FUNCTION_BLOCK FB_GC EXTENDS FB_PackMLModeSet
VAR_INPUT
	ServiceCtrl : REFERENCE TO ST_GC_ServiceCtrl;
	ServiceStatus : REFERENCE TO ST_GC_ServiceStatus;
	Admin : REFERENCE TO ST_GC_Admin;
	
	// Base unit used in GC chamber
	SpinAxis_BaseUnit : REFERENCE TO FB_AxisControl;
END_VAR

VAR_OUTPUT
	
END_VAR

VAR
	// 有需要特殊操作的需求，所以建立一個 ST_GC_ServiceCtrl 變數，讓程式內部可以過一手處理
	_ServiceCtrl : ST_GC_ServiceCtrl;
	_SpinAxisJogService : FB_GCSpinAxisJogServices;
	_SpinAxisMoveAbsService : FB_GCSpinAxisMoveAbsServices;
	_SpinAxisMoveVelService : FB_GCSpinAxisMoveVelServices;
END_VAR

A00_Service();
SUPER^();

ACTION A00_Service:
_SpinAxisJogService(
	Ctrl:= _ServiceCtrl.SpinAxisJog,
	Status:= ServiceStatus.SpinAxisJog,
	Axis_BaseUnit:= SpinAxis_BaseUnit,
	// Owner IDs are assigned by the Module so each Service instance is unique.
	ResourceOwnerId:= E_GCResourceOwnerId.SpinAxisJog);

_SpinAxisMoveAbsService(
	Ctrl:= _ServiceCtrl.SpinAxisMoveAbs,
	Status:= ServiceStatus.SpinAxisMoveAbs,
	Axis_BaseUnit:= SpinAxis_BaseUnit,
	ResourceOwnerId:= E_GCResourceOwnerId.SpinAxisMoveAbs);

_SpinAxisMoveVelService(
	Ctrl:= _ServiceCtrl.SpinAxisMoveVel,
	Status:= ServiceStatus.SpinAxisMoveVel,
	Axis_BaseUnit:= SpinAxis_BaseUnit,
	ResourceOwnerId:= E_GCResourceOwnerId.SpinAxisMoveVel);
END_ACTION

METHOD PROTECTED H_OnAborted
VAR_INPUT
	bFirstScan	: BOOL;
END_VAR
// Default action hook intentionally empty. Override in derived FBs when needed.
END_METHOD

METHOD PROTECTED H_OnAborting : E_PackMLHookResult
VAR_INPUT
	bFirstScan	: BOOL;
END_VAR
// Default transient hooks complete immediately; override when work is required.
H_OnAborting := E_PackMLHookResult.Done;
END_METHOD

METHOD PROTECTED H_OnClearing : E_PackMLHookResult
VAR_INPUT
	bFirstScan	: BOOL;
END_VAR
H_OnClearing := E_PackMLHookResult.Done;
END_METHOD

METHOD PROTECTED H_OnComplete
VAR_INPUT
	bFirstScan	: BOOL;
END_VAR
// Default action hook intentionally empty. Override in derived FBs when needed.
END_METHOD

METHOD PROTECTED H_OnCompleting : E_PackMLHookResult
VAR_INPUT
	bFirstScan	: BOOL;
END_VAR
// Default transient hooks complete immediately; override when work is required.
H_OnCompleting := E_PackMLHookResult.Done;
END_METHOD

METHOD PROTECTED H_OnExecute : E_PackMLHookResult
VAR_INPUT
	bFirstScan	: BOOL;
END_VAR
// Execute is stable by default; derived FBs decide when the process is done.
H_OnExecute := E_PackMLHookResult.Busy;

// Mapping control data
_ServiceCtrl := ServiceCtrl;
END_METHOD

METHOD PROTECTED H_OnHeld
VAR_INPUT
	bFirstScan	: BOOL;
END_VAR
// Default action hook intentionally empty. Override in derived FBs when needed.
END_METHOD

METHOD PROTECTED H_OnHolding : E_PackMLHookResult
VAR_INPUT
	bFirstScan	: BOOL;
END_VAR
// Default transient hooks complete immediately; override when work is required.
H_OnHolding := E_PackMLHookResult.Done;
END_METHOD

METHOD PROTECTED H_OnIdle
VAR_INPUT
	bFirstScan	: BOOL;
END_VAR
// Default action hook intentionally empty. Override in derived FBs when needed.
END_METHOD

METHOD PROTECTED H_OnModeChanged
VAR_INPUT
	ePreviousMode	: T_PackMLMode;
	eNewMode	: T_PackMLMode;
END_VAR
// Notice current mode to each service
_SpinAxisJogService.ModuleMode := eNewMode;
_SpinAxisMoveAbsService.ModuleMode := eNewMode;
_SpinAxisMoveVelService.ModuleMode := eNewMode;
END_METHOD

METHOD PROTECTED H_OnResetting : E_PackMLHookResult
VAR_INPUT
	bFirstScan	: BOOL;
END_VAR
H_OnResetting := E_PackMLHookResult.Busy;

// Request reset cmd to services
_ServiceCtrl.SpinAxisJog.Reset := TRUE;
_ServiceCtrl.SpinAxisMoveAbs.Reset := TRUE;
_ServiceCtrl.SpinAxisMoveVel.Reset := TRUE;

// Wait cmd finished
IF ServiceStatus.SpinAxisJog.State <> E_PackMLState.Idle
	OR ServiceStatus.SpinAxisMoveAbs.State <> E_PackMLState.Idle
	OR ServiceStatus.SpinAxisMoveVel.State <> E_PackMLState.Idle THEN
	RETURN;
END_IF

// Reset trigger
_ServiceCtrl.SpinAxisJog.Reset := FALSE;
_ServiceCtrl.SpinAxisMoveAbs.Reset := FALSE;
_ServiceCtrl.SpinAxisMoveVel.Reset := FALSE;

H_OnResetting := E_PackMLHookResult.Done;
END_METHOD

METHOD PROTECTED H_OnStarting : E_PackMLHookResult
VAR_INPUT
	bFirstScan	: BOOL;
END_VAR
// Default transient hooks complete immediately; override when work is required.
H_OnStarting := E_PackMLHookResult.Done;
END_METHOD

METHOD PROTECTED H_OnStopped
VAR_INPUT
	bFirstScan	: BOOL;
END_VAR
// Default action hook intentionally empty. Override in derived FBs when needed.
END_METHOD

METHOD PROTECTED H_OnStopping : E_PackMLHookResult
VAR_INPUT
	bFirstScan	: BOOL;
END_VAR
// Default transient hooks complete immediately; override when work is required.
H_OnStopping := E_PackMLHookResult.Done;
END_METHOD

METHOD PROTECTED H_OnSuspended
VAR_INPUT
	bFirstScan	: BOOL;
END_VAR
// Default action hook intentionally empty. Override in derived FBs when needed.
END_METHOD

METHOD PROTECTED H_OnSuspending : E_PackMLHookResult
VAR_INPUT
	bFirstScan	: BOOL;
END_VAR
// Default transient hooks complete immediately; override when work is required.
H_OnSuspending := E_PackMLHookResult.Done;
END_METHOD

METHOD PROTECTED H_OnUndefined : E_PackMLHookResult
VAR_INPUT
	bFirstScan	: BOOL;
END_VAR
// The base FB leaves Undefined immediately unless a derived FB delays startup.
H_OnUndefined := E_PackMLHookResult.Done;
END_METHOD

METHOD PROTECTED H_OnUnholding : E_PackMLHookResult
VAR_INPUT
	bFirstScan	: BOOL;
END_VAR
// Default transient hooks complete immediately; override when work is required.
H_OnUnholding := E_PackMLHookResult.Done;
END_METHOD

METHOD PROTECTED H_OnUnsuspending : E_PackMLHookResult
VAR_INPUT
	bFirstScan	: BOOL;
END_VAR
// Default transient hooks complete immediately; override when work is required.
H_OnUnsuspending := E_PackMLHookResult.Done;
END_METHOD

END_FUNCTION_BLOCK

(* stored: Version 1.1.0.1, ProductVersion 3.1.4026.18
   POU FB_GC: Id {d2b222b5-592d-46be-8a8e-fa50af509b93}, SpecialFunc None
   Folder StateAction: Id {92cfe23b-b998-4d76-8aa2-c8089e78aa61}
   Action A00_Service: Id {c62275db-aa76-4b4d-95ad-2ecb5851f919}
   Method H_OnAborted: Id {de8d6f56-427f-41df-b4d5-ddd289e1aed8}
   Method H_OnAborting: Id {29c05c7a-ae95-4991-b775-aae453451d8c}
   Method H_OnClearing: Id {b7069c3b-bd41-45c4-a177-00789e12f344}
   Method H_OnComplete: Id {9ab7169f-1450-41d3-b3d7-d608e72d68f0}
   Method H_OnCompleting: Id {6a295d34-cfdf-466f-b604-2e762f01df0b}
   Method H_OnExecute: Id {dc703a52-8c8a-4e2d-8deb-4adebb327ad6}
   Method H_OnHeld: Id {93f6b454-4398-4439-9237-4d01e13b7ccc}
   Method H_OnHolding: Id {d74d6d7d-e0fe-48fb-8a46-ad96f64e1fa5}
   Method H_OnIdle: Id {f9aa0f59-b1bb-45b6-82a2-3aac2bdc4e33}
   Method H_OnModeChanged: Id {9d68a966-aafb-43f3-857c-b18fd457d61a}
   Method H_OnResetting: Id {f6ec54bd-ad3d-49c4-9547-ff474beb3546}
   Method H_OnStarting: Id {2befc923-f5b2-4ef5-aa0b-77c9a7b33520}
   Method H_OnStopped: Id {ce5006a2-3926-4be3-8c7a-d8efdde1ca29}
   Method H_OnStopping: Id {2d9e9bf2-b821-4b2d-9e15-b22384f79334}
   Method H_OnSuspended: Id {cff92aa7-0bee-4d5f-a95f-be0ba263ee0f}
   Method H_OnSuspending: Id {5fe72161-6df8-45fc-8c16-29aa2466b4be}
   Method H_OnUndefined: Id {c8ca4bd2-e69c-48f1-bbc8-42b473d6b552}
   Method H_OnUnholding: Id {64c7cdee-7a16-4239-96a0-6ebcc2d0e61c}
   Method H_OnUnsuspending: Id {c36273cc-b3d2-484e-a95e-475cdbf1ae08} *)
